# EPICS substitutions: iocs/linkamIOC/linkamApp/Db/linkam.substitutions
# Macros:
#  P        PV Prefix for Linkam temp. controller
#  PORT     Asyn PORT
#  ADDR     Asyn ADDR
#  TIMEOUT  Asyn TIMEOUT
#  name     Template argument
file $(LINKAM3)/db/Linkam.template
{
pattern { P, PORT, ADDR, TIMEOUT, name }
    { "EA-LINKAM-01", "EA-LINKAM-01_AP", "0", "1", "LINKAM1" }
}

### Support for vacuum stages
#!file $(LINKAM3)/db/LinkamVacuum.template
#!{
#!pattern { P, PORT, ADDR, TIMEOUT, name }
#!    { "EA-LINKAM-01", "EA-LINKAM-01_AP", "0", "1", "LINKAM1" }
#!}

### Support for the RHGen (humidity stages)
#!file $(LINKAM3)/db/LinkamRHGen.template
#!{
#!pattern { P, PORT, ADDR, TIMEOUT, name }
#!    { "EA-LINKAM-01", "EA-LINKAM-01_AP", "0", "1", "LINKAM1" }
#!}
